(* Logix 5000 project; controller Uidaho_Factory vendor 1 type 14 code 165 rev 38.11; software revision 38.00; part 3 of 3 *)
(* tags used below, declared in another part *)
   SLD_start : DINT;
   SSC_start : DINT;
   VGR_start : DINT;
   PWM_Outputs : PWM_Out[20];
(* MainProgram, continued *)

ROUTINE Test_SLD   (* ladder *)
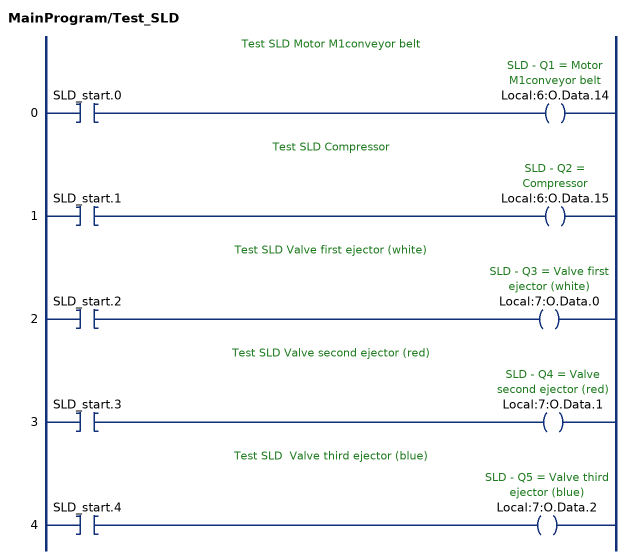
   // Test SLD Motor M1conveyor belt
   0: XIC(SLD_start.0)OTE(Local:6:O.Data.14);
   // Test SLD Compressor
   1: XIC(SLD_start.1)OTE(Local:6:O.Data.15);
   // Test SLD Valve first ejector (white)
   2: XIC(SLD_start.2)OTE(Local:7:O.Data.0);
   // Test SLD Valve second ejector (red)
   3: XIC(SLD_start.3)OTE(Local:7:O.Data.1);
   // Test SLD  Valve third ejector (blue)
   4: XIC(SLD_start.4)OTE(Local:7:O.Data.2);
END_ROUTINE

ROUTINE Test_SSC   (* ladder *)
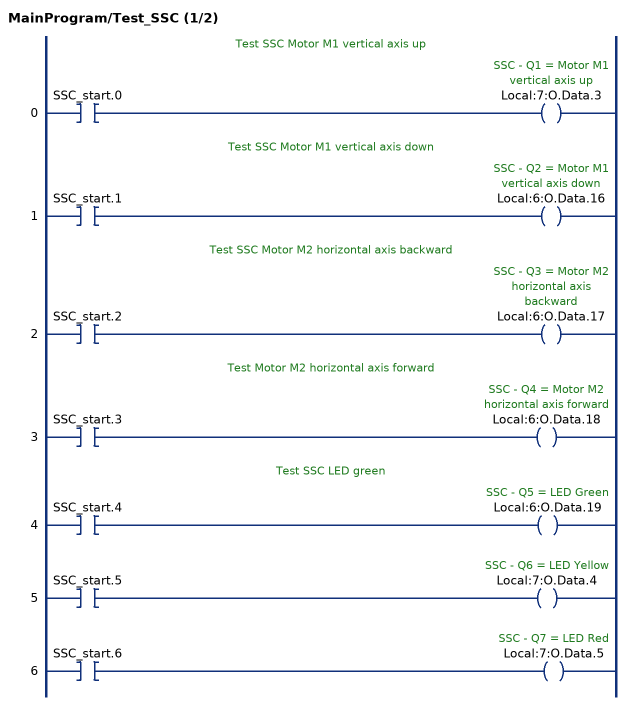
   // Test SSC Motor M1 vertical axis up
   0: XIC(SSC_start.0)OTE(Local:7:O.Data.3);
   // Test SSC Motor M1 vertical axis down
   1: XIC(SSC_start.1)OTE(Local:6:O.Data.16);
   // Test SSC Motor M2 horizontal axis backward
   2: XIC(SSC_start.2)OTE(Local:6:O.Data.17);
   // Test Motor M2 horizontal axis forward
   3: XIC(SSC_start.3)OTE(Local:6:O.Data.18);
   // Test SSC LED green
   4: XIC(SSC_start.4)OTE(Local:6:O.Data.19);
   5: XIC(SSC_start.5)OTE(Local:7:O.Data.4);
   6: XIC(SSC_start.6)OTE(Local:7:O.Data.5);
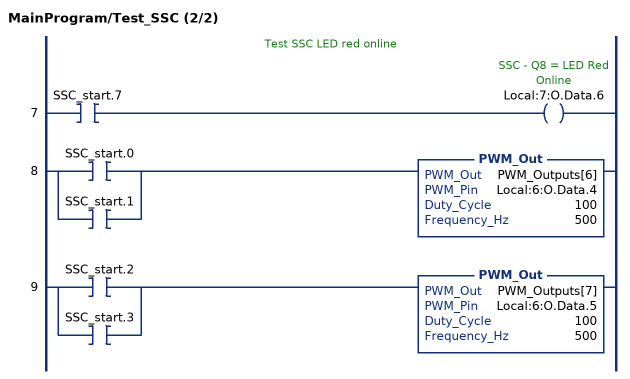
   // Test SSC LED red online
   7: XIC(SSC_start.7)OTE(Local:7:O.Data.6);
   8: [XIC(SSC_start.0) ,XIC(SSC_start.1) ]PWM_Out(PWM_Outputs[6],Local:6:O.Data.4,100,500);
   9: [XIC(SSC_start.2) ,XIC(SSC_start.3) ]PWM_Out(PWM_Outputs[7],Local:6:O.Data.5,100,500);
END_ROUTINE

ROUTINE Test_VGR   (* ladder *)
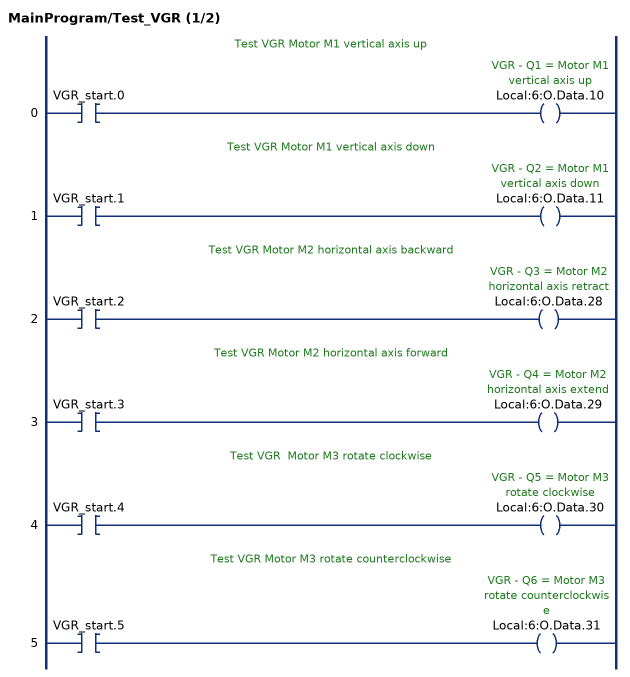
   // Test VGR Motor M1 vertical axis up
   0: XIC(VGR_start.0)OTE(Local:6:O.Data.10);
   // Test VGR Motor M1 vertical axis down
   1: XIC(VGR_start.1)OTE(Local:6:O.Data.11);
   // Test VGR Motor M2 horizontal axis backward
   2: XIC(VGR_start.2)OTE(Local:6:O.Data.28);
   // Test VGR Motor M2 horizontal axis forward
   3: XIC(VGR_start.3)OTE(Local:6:O.Data.29);
   // Test VGR  Motor M3 rotate clockwise
   4: XIC(VGR_start.4)OTE(Local:6:O.Data.30);
   // Test VGR Motor M3 rotate counterclockwise
   5: XIC(VGR_start.5)OTE(Local:6:O.Data.31);
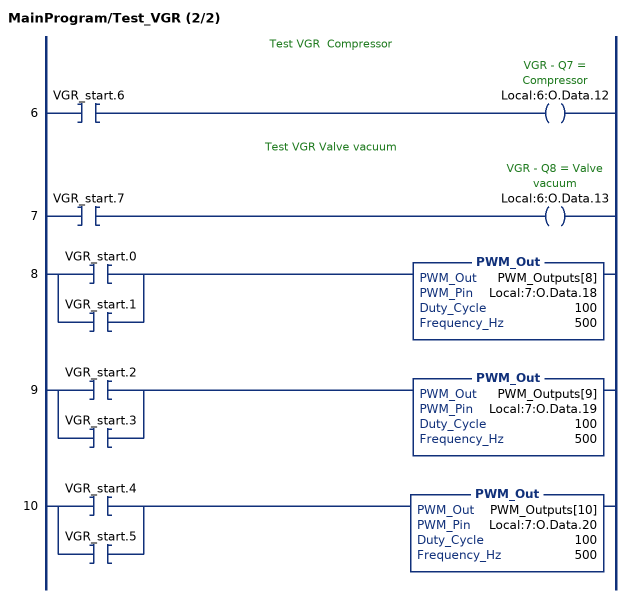
   // Test VGR  Compressor
   6: XIC(VGR_start.6)OTE(Local:6:O.Data.12);
   // Test VGR Valve vacuum
   7: XIC(VGR_start.7)OTE(Local:6:O.Data.13);
   8: [XIC(VGR_start.0) ,XIC(VGR_start.1) ]PWM_Out(PWM_Outputs[8],Local:7:O.Data.18,100,500);
   9: [XIC(VGR_start.2) ,XIC(VGR_start.3) ]PWM_Out(PWM_Outputs[9],Local:7:O.Data.19,100,500);
   10: [XIC(VGR_start.4) ,XIC(VGR_start.5) ]PWM_Out(PWM_Outputs[10],Local:7:O.Data.20,100,500);
END_ROUTINE
END_PROGRAM
